FUNCTION_BLOCK FB_MotionInterlocks IMPLEMENTS I_MotionInterlocks
VAR_INPUT
END_VAR
VAR_OUTPUT
END_VAR
VAR
    {attribute 'hide'}
    iMotionLogger 		: I_MotionLogger;
    {attribute 'hide'}
    iMotionInterlocksShareData : I_MotionInterlocksShareData;
    {attribute 'hide'}
    bAllForwardEnabled: BOOL:=FALSE;
    // Backward enable EPS summary
    {attribute 'hide'}
    bAllBackwardEnabled: BOOL:=FALSE;
    {attribute 'hide'}
    {attribute 'hide'}
    bAllEnabled: BOOL:=FALSE;
   // If TRUE, we want to enable the motor independently of PMPS or other safety systems.
    bPowerSelf: BOOL:=FALSE;
    // TRUE if we have safety permission to move
    bSafetyReady: BOOL;
   // NC STO Input: TRUE if ok to move
    {attribute 'pytmc' := '
        pv: PLC:bHardwareEnable
        io: i
        field: ZNAM FALSE
        field: ONAM TRUE
        field: DESC TRUE if STO not hit
    '}
    bHardwareEnable AT %I*: BOOL ;

    // Used by the IOC to disable an axis
    {attribute 'pytmc' := '
        pv: PLC:bUserEnable
        io: io
        field: ZNAM DISABLE
        field: ONAM ENABLE
        field: DESC Used to disable power entirely for an axis
    '}
    bUserEnable: BOOL := TRUE;
    {attribute 'hide'}
    bHomeBusy : BOOL;
    {attribute 'hide'}
    bMoveBusy	: BOOL;
    {attribute 'hide'}
    bNewMoveReq	: BOOL;
    {attribute 'hide'}
    bEnable: BOOL;
    {attribute 'hide'}
    bExecute : BOOL;
    {attribute 'hide'}
    sMessage : STRING;
    {attribute 'hide'}
    bWarning : BOOL;
    {attribute 'hide'}
    nErpicsWarnId : UINT;
    {attribute 'hide'}
    bError : BOOL;
    {attribute 'hide'}
    nErrorID : BOOL;
    {attribute 'hide'}
    bReset : BOOL;
    {attribute 'hide'}
    bMoveOk : BOOL;
END_VAR

IF ( iMotionInterlocksShareData = 0 ) OR ( iMotionLogger = 0) THEN
    // throw an exception
    RETURN;
END_IF

// read share
bAllEnabled := iMotionInterlocksShareData.DriveEnable AND bHardwareEnable;
bAllEnabled R= NOT bUserEnable;
// Moves are automatically allowed if no safety hooks. Otherwise, some other code will set this.
bSafetyReady S= bPowerSelf;

IF NOT bUserEnable THEN
    bError := TRUE;
    nErrorID:= 1;
    bMoveOk := FALSE;
    sMessage := 'User enable interlock triggered!';
ELSIF NOT bHardwareEnable THEN
    bError := TRUE;
    nErrorID:= 1;
    bMoveOk := FALSE;
    sMessage := 'Hardware enbale interlocks triggered!';
END_IF

// wait for global reset event to complete
bReset := iMotionInterlocksShareData.ResetDone;
IF bReset THEN
    bReset := FALSE;
    bError := FALSE;
    bWarning := FALSE;
    nErrorID:= 0;
    sMessage:='';
END_IF

//FB_Init is always available implicitly and it is used primarily for initialization.
//The return value is not evaluated. For a specific influence, you can also declare the
//methods explicitly and provide additional code there with the standard initialization
//code. You can evaluate the return value.
METHOD FB_Init: BOOL
VAR_INPUT
    bInitRetains: BOOL; // TRUE: the retain variables are initialized (reset warm / reset cold)
    bInCopyCode: BOOL;  // TRUE: the instance will be copied to the copy code afterward (online change)

    iMotionLogger 		: I_MotionLogger;
    iMotionInterlocksShareData : I_MotionInterlocksShareData;
END_VAR
THIS^.iMotionLogger := iMotionLogger;
THIS^.iMotionInterlocksShareData := iMotionInterlocksShareData;
END_METHOD

{warning 'Add property implementation'}
PROPERTY InterlocksError : BOOL
GET
END_GET
END_PROPERTY

{warning 'Add property implementation'}
PROPERTY InterlocksErrorID : UDINT
GET
END_GET
END_PROPERTY

{warning 'Add property implementation'}
PROPERTY InterlocksErrorMessage : STRING
GET
END_GET
END_PROPERTY

{warning 'Add property implementation'}
PROPERTY MoveBackwardEnabled : BOOL
GET
END_GET
END_PROPERTY

{warning 'Add property implementation'}
PROPERTY MoveForwardEnabled : BOOL
GET
END_GET
END_PROPERTY

{warning 'Add method implementation '}
METHOD MoveOk : BOOL
VAR_INPUT
    NewMoveReq	: BOOL;
    Enable	: BOOL;
    Execute	: BOOL;
END_VAR
END_METHOD

{warning 'Add property implementation'}
PROPERTY PowerEnabled : BOOL
GET
END_GET
END_PROPERTY

END_FUNCTION_BLOCK

(* stored: Version 1.1.0.1
   POU FB_MotionInterlocks: Id {b69073ed-2a55-41fc-84a9-b8fe79332e5e}, SpecialFunc None
   Method FB_Init: Id {ee1048d7-3a0b-4701-a887-c2bc01c18e00}
   Property InterlocksError: Id {0e139e64-82f7-44db-b026-c8b3a3ce7de8}
   Get Get: Id {3d402358-4896-4b22-86f8-09f4d880f427}
   Property InterlocksErrorID: Id {dc1898a9-f714-4f91-b9c5-eb1143afddd3}
   Get Get: Id {acbadcd5-5050-4f73-a022-6b7291e0c444}
   Property InterlocksErrorMessage: Id {3c6151d2-7e95-4fde-9e74-00243a7324b7}
   Get Get: Id {36059109-c6c7-449c-9aad-333c51d4e917}
   Property MoveBackwardEnabled: Id {73228441-2498-4cbf-b7a0-4009813e3963}
   Get Get: Id {f4731fcf-cdb2-4505-9bf3-b0970507bbd1}
   Property MoveForwardEnabled: Id {dbd2e5c0-7ee3-4d69-bfac-0c4778db19bb}
   Get Get: Id {b2fba177-14e5-4ae4-b487-6f6969050bec}
   Method MoveOk: Id {3c80f11d-c026-4b06-9cfb-6a7a45c3d176}
   Property PowerEnabled: Id {6a435248-a266-41ef-9b9c-8e0bf7663a4b}
   Get Get: Id {c27ac7b3-d93e-4dca-97d4-f9f71a18aff4} *)
